(* Logix 5000 project; controller CarbonScout_MK6 vendor 1 type 14 code 154 rev 32.11; software revision 32.00; part 2 of 17 *)
(* tags used below, declared in another part *)
   Inp_PV : REAL;   // Input Signal (process variable) from Sensor
   Inp_PVSrcQ : DINT;   // Input Source and Quality (from Channel object, if available) (enum)
   Inp_PVBad : BOOL;   // 1=PV or I/O Comms Status Bad, 0=OK
   Inp_PVUncertain : BOOL;   // 1=PV Value Not Reliable, 0=OK
   Inp_Sim : BOOL;   // 1=Use simulated PV (Set_SimPV); 0=Use Input (Inp_PV)
   Inp_Reset : BOOL;   // 1=Reset all Alarms requiring reset
   Cfg_NoSubstPV : BOOL;   // 1=Disallow selection of Substitute PV
   Cfg_SetTrack : BOOL;   // 1=PSets track OSets in Oper, OSets track PSets in Prog, 0=no tracking
   Cfg_HasChanObj : BOOL;   // 1=Tells HMI a Channel object (AIChan, etc.) is used for Inp_PV
   Cfg_UseChanSrcQ : BOOL;   // 1=Pass thru connected Channel's SrcQ value, 0=generate SrcQ
   Cfg_PCmdClear : ALIAS FOR Mode.Cfg_PCmdClear;
   Cfg_InpRawMin : REAL;   // Input (unscaled) Minimum for Scaling
   Cfg_InpRawMax : REAL;   // Input (unscaled) Maximum for Scaling
   Cfg_PVEUMin : REAL;   // PV (Output) Minimum for Scaling to EU
   Cfg_PVEUMax : REAL;   // PV (Output) Maximum for Scaling to EU
   Cfg_FiltTC : REAL;   // PV Filter Time Constant (s), 0.0 = unfiltered
   Cfg_HiHiDB : REAL;   // High-High Status Deadband (EU)
   Cfg_HiDB : REAL;   // High Status Deadband (EU)
   Cfg_LoDB : REAL;   // Low Status Deadband (EU)
   Cfg_LoLoDB : REAL;   // Low-Low Status Deadband (EU)
   Cfg_FailHiLim : REAL;   // Out-of-Range (fail) High Limit (EU)
   Cfg_FailLoLim : REAL;   // Out-of-Range (fail) Low Limit (EU)
   Cfg_FailDB : REAL;   // Out-of-Range (fail) High/Low Deadband (EU)
   PSet_Owner : DINT;   // Program Owner Request ID (non-zero) or Release (zero)
   PSet_HiHiLim : REAL;   // Program-Entered High-High Status Threshold (EU)
   PSet_HiLim : REAL;   // Program-Entered High Status Threshold (EU)
   PSet_LoLim : REAL;   // Program-Entered Low Status Threshold (EU)
   PSet_LoLoLim : REAL;   // Program-Entered Low-Low Status Threshold (EU)
   MSet_SubstPV : REAL;   // Maintenance-Entered Substitute PV (EU)
   OSet_HiHiLim : REAL;   // Operator-Entered High-High Status Threshold (EU)
   OSet_HiLim : REAL;   // Operator-Entered High Status Threshold (EU)
   OSet_LoLim : REAL;   // Operator-Entered Low Status Threshold (EU)
   OSet_LoLoLim : REAL;   // Operator-Entered Low-Low Status Threshold (EU)
   Set_SimPV : REAL;   // PV used in Simulation (Inp_Sim=1) (EU)
   PCmd_ClearCapt : BOOL;   // Program Command to Clear the captured min / max PV excursion values
   PCmd_Reset : BOOL;   // Program Command to Reset all Alarms requiring Reset
   PCmd_HiHiAck : ALIAS FOR HiHi.PCmd_Ack;   // Program Command to Acknowledge High-High Alarm
   PCmd_HiAck : ALIAS FOR Hi.PCmd_Ack;   // Program Command to Acknowledge High Alarm
   PCmd_LoAck : ALIAS FOR Lo.PCmd_Ack;   // Program Command to Acknowledge Low Alarm
   PCmd_LoLoAck : ALIAS FOR LoLo.PCmd_Ack;   // Program Command to Acknowledge Low-Low Alarm
   PCmd_FailAck : ALIAS FOR Fail.PCmd_Ack;   // Program Command to Acknowldege Analog Input Failure Alarm
   MCmd_SubstPV : BOOL;   // Maintenance Command to use Substitute PV (override input)
   MCmd_InpPV : BOOL;   // Maintenance Command to use Input PV (normal)
   OCmd_ClearCapt : BOOL;   // Operator Command to Clear the captured min / max PV excursion values
   OCmd_Reset : BOOL;   // Operator Command to Reset all Alarms requiring Reset
   OCmd_ResetAckAll : BOOL;   // Operator Command to Reset and Acknowledge all Alarms
   Val : REAL;   // Analog Value (after Substitute PV, if used)
   Val_InpPV : REAL;   // Analog Input Value (actual, before Substitute PV selection)
   Val_PVMinCapt : REAL;   // Captured PV Minimum (excursion) since last cleared
   Val_PVMaxCapt : REAL;   // Captured PV Maximum (excursion) since last cleared
   Val_PVEUMin : REAL;   // Minimum of scaled range = MIN (Cfg_PVEUMin, Cfg_PVEUMax)
   Val_PVEUMax : REAL;   // Maximum of scaled range = MAX (Cfg_PVEUMin, Cfg_PVEUMax)
   SrcQ_IO : DINT;   // Source and Quality of primary I/O (enumeration)
   SrcQ : DINT;   // Source and Quality of primary Val/Sts (enumeration)
   Val_Fault : DINT;   // Device Fault Status 0=none, 20=Lo, 21=Hi, 24=LoLo, 25=HiHi, 32=Fail, 34=CfgErr
   Val_Owner : DINT;   // Current Object Owner ID (0=not owned)
   Val_Notify : DINT;   // Current Alarm Level and Acknowledgement (enumeration)
   Val_HiHiLim : REAL;   // Current High-High Status Threshold
   Val_HiLim : REAL;   // Current High Status Threshold
   Val_LoLim : REAL;   // Current Low Status Threshold
   Val_LoLoLim : REAL;   // Current Low-Low Status Threshold
   Sts_SubstPV : BOOL;   // 1=Using Substitute PV (Input being overridden)
   Sts_InpPV : BOOL;   // 1=Using Input PV (normal)
   Sts_PVBad : BOOL;   // 1=PV Bad quality or Out of Range
   Sts_PVUncertain : BOOL;   // 1=PV Value is Uncertain (quality)
   Sts_MaintByp : BOOL;   // 1=A Maintenance Bypass is Active, display icon
   Sts_AlmInh : BOOL;   // 1=An Alarm is Shelved, Disabled or Suppressed: display icon
   Sts_Err : BOOL;   // 1=Error in Config (see detail Err_ bits for reason), display icon
   Err_Raw : BOOL;   // 1=Error in Config: Raw Input Scaling Min = Max
   Err_EU : BOOL;   // 1=Error in Config: Scaled EU Min = Max
   Err_Timer : BOOL;   // 1=Error in Config: On Delay, Off Delay, Gate Delay Time Invalid (use 0 to 2147483 s)
   Err_Filt : BOOL;   // 1=Error in Config: PV filter params (RateTime, TC)
   Err_DB : BOOL;   // 1=Error in Config: a Status Deadband is < 0.0
   Err_Alarm : BOOL;   // 1=Error in Config: Alarm Min On Time, Shelf Time, Severity
   Sts_Maint : ALIAS FOR Mode.Sts_Maint;
   Sts_Prog : ALIAS FOR Mode.Sts_Prog;
   Sts_Oper : ALIAS FOR Mode.Sts_Oper;
   Sts_HiHiCmp : ALIAS FOR HiHiGate.Inp;   // PV High-High comparison result 1=High-High
   Sts_HiHi : ALIAS FOR HiHi.Inp;   // 1=Analog Input is above High-High limit
   Sts_HiCmp : ALIAS FOR HiGate.Inp;   // PV High comparison result 1=High
   Sts_Hi : ALIAS FOR Hi.Inp;   // 1=Analog Input is above High limit
   Sts_LoCmp : ALIAS FOR LoGate.Inp;   // PV Low comparison result 1=Low
   Sts_Lo : ALIAS FOR Lo.Inp;   // 1=Analog Input is below Low limit
   Sts_LoLoCmp : ALIAS FOR LoLoGate.Inp;   // PV Low-Low comparison result 1=Low-Low
   Sts_LoLo : ALIAS FOR LoLo.Inp;   // 1=Analog Input is below Low-Low limit
   Sts_FailCmp : ALIAS FOR FailGate.Inp;   // PV Fail comparison result 1=Out of Range
   Sts_Fail : ALIAS FOR Fail.Inp;   // 1=Analog Input is Out of Range or PV Bad
   Rdy_SubstPV : BOOL;   // 1=Ready for MCmd_SubstPV
   Rdy_InpPV : BOOL;   // 1=Ready for MCmd_InpPV
   Rdy_OSet : BOOL;   // 1=Ready to receive OSets (enables data entry fields)
   P_AIn : BOOL;   // Unique Parameter Name for auto - discovery
   LoLo : P_Alarm;   // Low-Low Alarm
   Lo : P_Alarm;   // Low Alarm
   Hi : P_Alarm;   // High Alarm
   HiHi : P_Alarm;   // High-High Alarm
   Mode : P_Mode;   // Analog Input Mode Selection
   Cfg_Tag : STRING_12;   // Tagname for display on HMI
   Cfg_Label : STRING_12;   // Label for graphic symbol displayed on HMI
   Cfg_Desc : STRING_20;   // Description for display on HMI
   Fail : P_Alarm;   // Analog Input Failure Alarm (bad quality or out of range)
   Wrk_Notify : DINT;   // Buffer for building Val_Notify
   Wrk_SrcQ : DINT;   // Register for building Source / Quality enumeration
   Wrk_Fault : DINT;   // Buffer for building Val_Fault
   Wrk_SubstPV : BOOL;   // Internal flag: Using Substitute PV
   Wrk_UnfiltPV : REAL;   // Unfiltered PV, input to 1st order filter
   Wrk_Alpha : REAL;   // Filter multiplier = (1 / (1+TC/dT) )
   Wrk_ScanT : TIMER;   // Scan Timer (milliseconds, always runs)
   Wrk_ScanTime : REAL;   // Time since this instance was last scanned
   Wrk_FiltPV : REAL;   // Filtered PV
   Wrk_ValidONS : BOOL;   // Selected PV goes from Infinite or Not a Number to VALID
   Wrk_SelPVDINT : DINT;   // Selected PV check for Infinite or Non A Number
   Wrk_SelPVInfNaN : BOOL;   // Selected PV (Input or Substitute) is Infinite or NaN
   Wrk_Fail : BOOL;   // Internal flag: Fail Status
   Wrk_LoLo : BOOL;   // Internal flag: Low-Low Status
   Wrk_Lo : BOOL;   // Internal flag: Low Status
   Wrk_Hi : BOOL;   // Internal flag: High Status
   Wrk_HiHi : BOOL;   // Internal flag: High-High Status
   FailGate : P_Gate;   // Fail Alarm Gate / Delay Block
   LoLoGate : P_Gate;   // Low-Low Alarm Gate / Delay Block
   LoGate : P_Gate;   // Low Alarm Gate / Delay Block
   HiHiGate : P_Gate;   // High-High Alarm Gate / Delay Block
   HiGate : P_Gate;   // High Alarm Gate / Delay Block
   Wrk_InpInfNaN : BOOL;   // Input is Infinite or Not a Number
   Wrk_InpDINT : DINT;   // Input REAL bit pattern as a DINT (check for Inf/NaN)
   Wrk_InpFail : BOOL;   // Input Fail: out of range
   Simulation : DINT;
   test : DINT;
(* P_AIn, continued *)

ROUTINE Logic   (* ladder *)
// Normal Scan - PV is scaled and alarms are generated
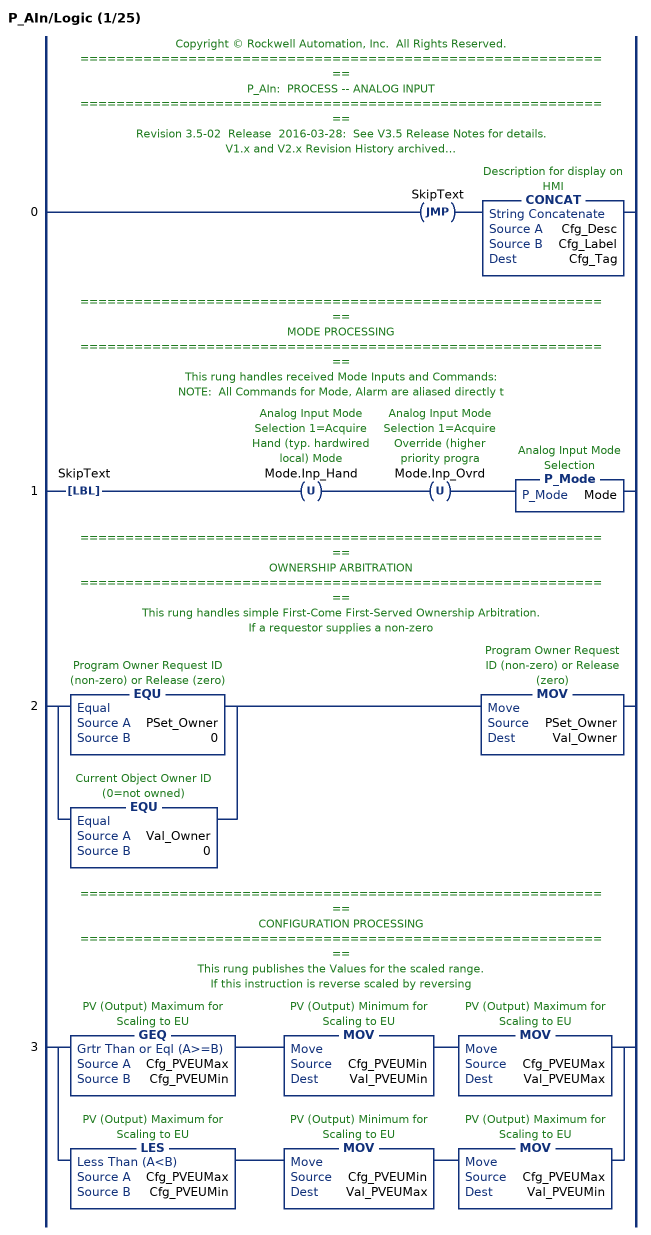
   // Copyright © Rockwell Automation, Inc.  All Rights Reserved.
   // ============================================================
   // P_AIn:  PROCESS -- ANALOG INPUT
   // ============================================================
   // Revision 3.5-02  Release  2016-03-28:  See V3.5 Release Notes for details.
   // V1.x and V2.x Revision History archived.
   // V3.0-00  2013-06-30:  Uses P_Gate, P_Alarm, P_Mode V3.0.
   // Added Inf_Lib, navigation to Channel obj.
   // V3.0-01  2013-07-30:  Modified Parameter descriptions only.
   // V3.0-02  2013-09-03:  Modified Parameter descriptions only.
   // V3.0-03  2013-10-30:  Corrected Parameter descriptions and default
   // configuration values for alarms only.
   // V3.0-04  2014-04-04:   Improved handling of Inf/NaN to avoid Minor Faults.
   // V3.1-00  2014-07-08:  Modified to use P_Alarm, P_Mode V3.1, add SrcQ enums.
   // Modified to consistently use alias tag names.
   // V3.1-01  2014-09-03:  Inp_PVSrcQ pulled into all bad/uncertain logic.
   // Using P_Alarm, P_Gate, P_Mode V3.1-01.
   // V3.1-02  2014-09-30:  Unchanged, but using P_Alarm V3.1-02.
   // V3.1-05  2016-01-22:  Added check of SrcQ >= 32 for Val_Fault.
   // Changed default values of min, max capture. Modified to
   // handle on-delay near status thresholds properly.
   // V3.5-01  2016-01-29:  Unchanged, using P_Alarm, P_Gate V3.5-01.
   // V3.5-02  2016-03-28:  Added Cfg_UseChanSrcQ to make SrcQ use
   // independent of Cfg_HasChanObj, which is for navigation only.
   // ============================================================
   // This Instruction monitors an Analog Input from a flow, level, pressure,
   // temperature, or any other analog sensor, and provides:
   // *  Scaling, from Input (Raw) to PV (Engineering) Units
   // *  High-High, High, Low and Low-Low Status and Alarms, with Gate
   // inputs and configurable on-delay, off-delay and gate delay times
   // *  Monitoring of bad/uncertain PV status, floating point exceptions
   // and out-of-range conditions, with PV Fail alarm
   // *  Setting of a simulated input signal for process simulation
   // *  Capturing of the lowest and highest PV excursion values
   // *  Program and Operator Settings for Status Thresholds
   // *  Configurable threshold deadbands and out of range limits
   // *  Maintenance Commands to allow manual override of the input signal (Substitute PV)
   // Modes are provided by a P_Mode AOI instance.
   // Alarms are provided by P_Alarm AOI instances.
   // Status gating provided by P_Gate AOI instances.
   // Modes of operation: Operator, Program, Maintenance
   // ============================================================
   // SHOW LOCAL STRINGS
   // ============================================================
   // The STRINGs containing the text associated with each instance of this
   // instruction cannot be Input or Output Parameters, because STRINGs are not
   //  'atomic' types. (Inputs and Outputs must be SINT, INT, DINT, REAL, or BOOL.)
   // In order to make it easier to find and configure these STRINGs, this rung
   // was added.  THE JMP (and the LBL on the following rung)
   // MUST NOT BE REMOVED!!!
   // To view the STRINGs, go to the instruction instance (in LD or FBD), RIGHT-click
   // to bring up the context menu and select "Open Instruction Logic".
   // This rung will appear with the STRING values for the selected instance.
   // You may double-click the STRING values here to modify them as well.
   // #####  V3.0-00  2013-06-30:  Added Inf_Lib  #####
   0: JMP(SkipText)CONCAT(Cfg_Desc,Cfg_Label,Cfg_Tag);
   // ============================================================
   // MODE PROCESSING
   // ============================================================
   // This rung handles received Mode Inputs and Commands:
   // NOTE:  All Commands for Mode, Alarm are aliased directly t
   1: LBL(SkipText)OTU(Mode.Inp_Hand)OTU(Mode.Inp_Ovrd)P_Mode(Mode);
   // ============================================================
   // OWNERSHIP ARBITRATION
   // ============================================================
   // This rung handles simple First-Come First-Served Ownership Arbitration.
   // If a requestor supplies a non-zero
   2: [EQU(PSet_Owner,0) ,EQU(Val_Owner,0) ]MOV(PSet_Owner,Val_Owner);
   // ============================================================
   // CONFIGURATION PROCESSING
   // ============================================================
   // This rung publishes the Values for the scaled range.
   // If this instruction is reverse scaled by reversing
   3: [GEQ(Cfg_PVEUMax,Cfg_PVEUMin) MOV(Cfg_PVEUMin,Val_PVEUMin) MOV(Cfg_PVEUMax,Val_PVEUMax) ,LES(Cfg_PVEUMax,Cfg_PVEUMin) MOV(Cfg_PVEUMin,Val_PVEUMax) MOV(Cfg_PVEUMax,Val_PVEUMin) ];
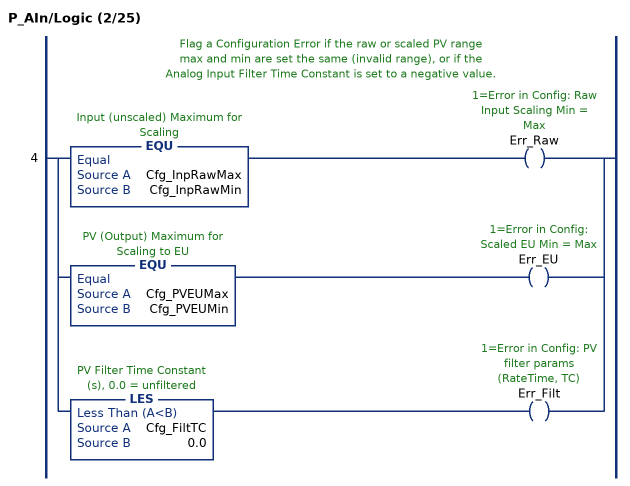
   // Flag a Configuration Error if the raw or scaled PV range
   // max and min are set the same (invalid range), or if the
   // Analog Input Filter Time Constant is set to a negative value.
   4: [EQU(Cfg_InpRawMax,Cfg_InpRawMin) OTE(Err_Raw) ,EQU(Cfg_PVEUMax,Cfg_PVEUMin) OTE(Err_EU) ,LES(Cfg_FiltTC,0.0) OTE(Err_Filt) ];
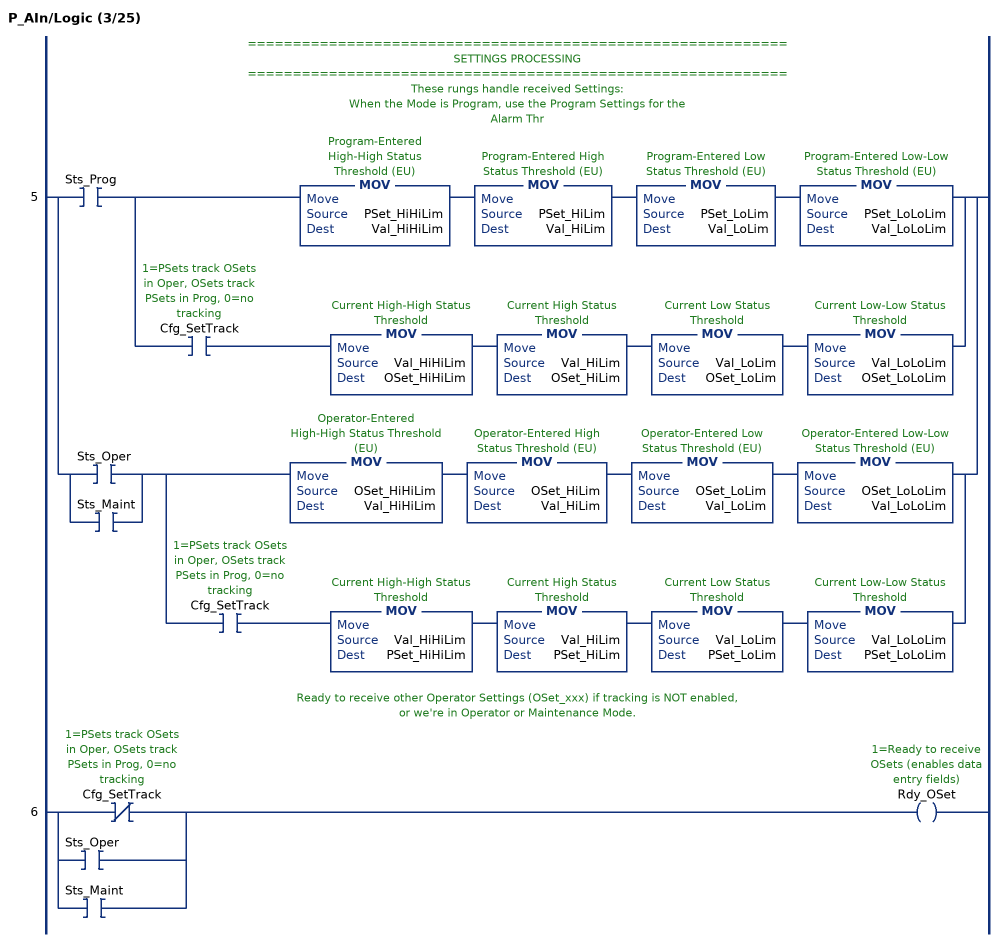
   // ============================================================
   // SETTINGS PROCESSING
   // ============================================================
   // These rungs handle received Settings:
   // When the Mode is Program, use the Program Settings for the
   // Alarm Thr
   5: [XIC(Sts_Prog) [MOV(PSet_HiHiLim,Val_HiHiLim) MOV(PSet_HiLim,Val_HiLim) MOV(PSet_LoLim,Val_LoLim) MOV(PSet_LoLoLim,Val_LoLoLim) ,XIC(Cfg_SetTrack) MOV(Val_HiHiLim,OSet_HiHiLim) MOV(Val_HiLim,OSet_HiLim) MOV(Val_LoLim,OSet_LoLim) MOV(Val_LoLoLim,OSet_LoLoLim) ] ,[XIC(Sts_Oper) ,XIC(Sts_Maint) ] [MOV(OSet_HiHiLim,Val_HiHiLim) MOV(OSet_HiLim,Val_HiLim) MOV(OSet_LoLim,Val_LoLim) MOV(OSet_LoLoLim,Val_LoLoLim) ,XIC(Cfg_SetTrack) MOV(Val_HiHiLim,PSet_HiHiLim) MOV(Val_HiLim,PSet_HiLim) MOV(Val_LoLim,PSet_LoLim) MOV(Val_LoLoLim,PSet_LoLoLim) ] ];
   // Ready to receive other Operator Settings (OSet_xxx) if tracking is NOT enabled,
   // or we're in Operator or Maintenance Mode.
   6: [XIO(Cfg_SetTrack) ,XIC(Sts_Oper) ,XIC(Sts_Maint) ]OTE(Rdy_OSet);
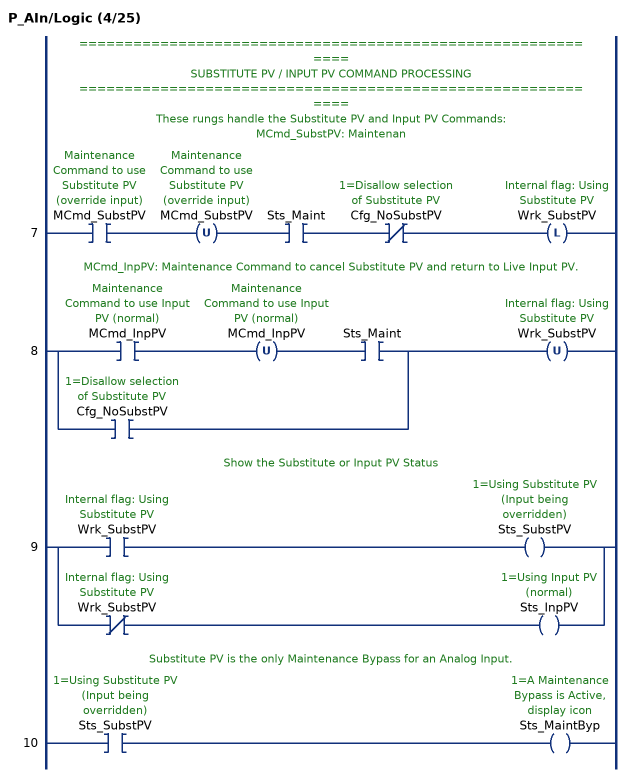
   // ============================================================
   // SUBSTITUTE PV / INPUT PV COMMAND PROCESSING
   // ============================================================
   // These rungs handle the Substitute PV and Input PV Commands:
   // MCmd_SubstPV: Maintenan
   7: XIC(MCmd_SubstPV)OTU(MCmd_SubstPV)XIC(Sts_Maint)XIO(Cfg_NoSubstPV)OTL(Wrk_SubstPV);
   // MCmd_InpPV: Maintenance Command to cancel Substitute PV and return to Live Input PV.
   8: [XIC(MCmd_InpPV) OTU(MCmd_InpPV) XIC(Sts_Maint) ,XIC(Cfg_NoSubstPV) ]OTU(Wrk_SubstPV);
   // Show the Substitute or Input PV Status
   9: [XIC(Wrk_SubstPV) OTE(Sts_SubstPV) ,XIO(Wrk_SubstPV) OTE(Sts_InpPV) ];
   // Substitute PV is the only Maintenance Bypass for an Analog Input.
   10: XIC(Sts_SubstPV)OTE(Sts_MaintByp);
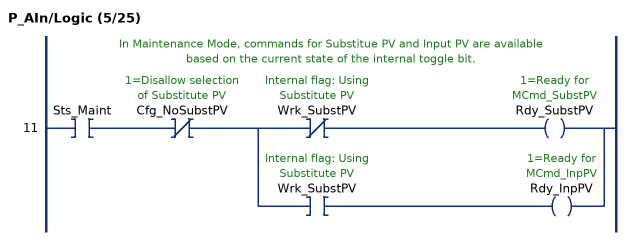
   // In Maintenance Mode, commands for Substitue PV and Input PV are available
   // based on the current state of the internal toggle bit.
   11: XIC(Sts_Maint)XIO(Cfg_NoSubstPV)[XIO(Wrk_SubstPV) OTE(Rdy_SubstPV) ,XIC(Wrk_SubstPV) OTE(Rdy_InpPV) ];
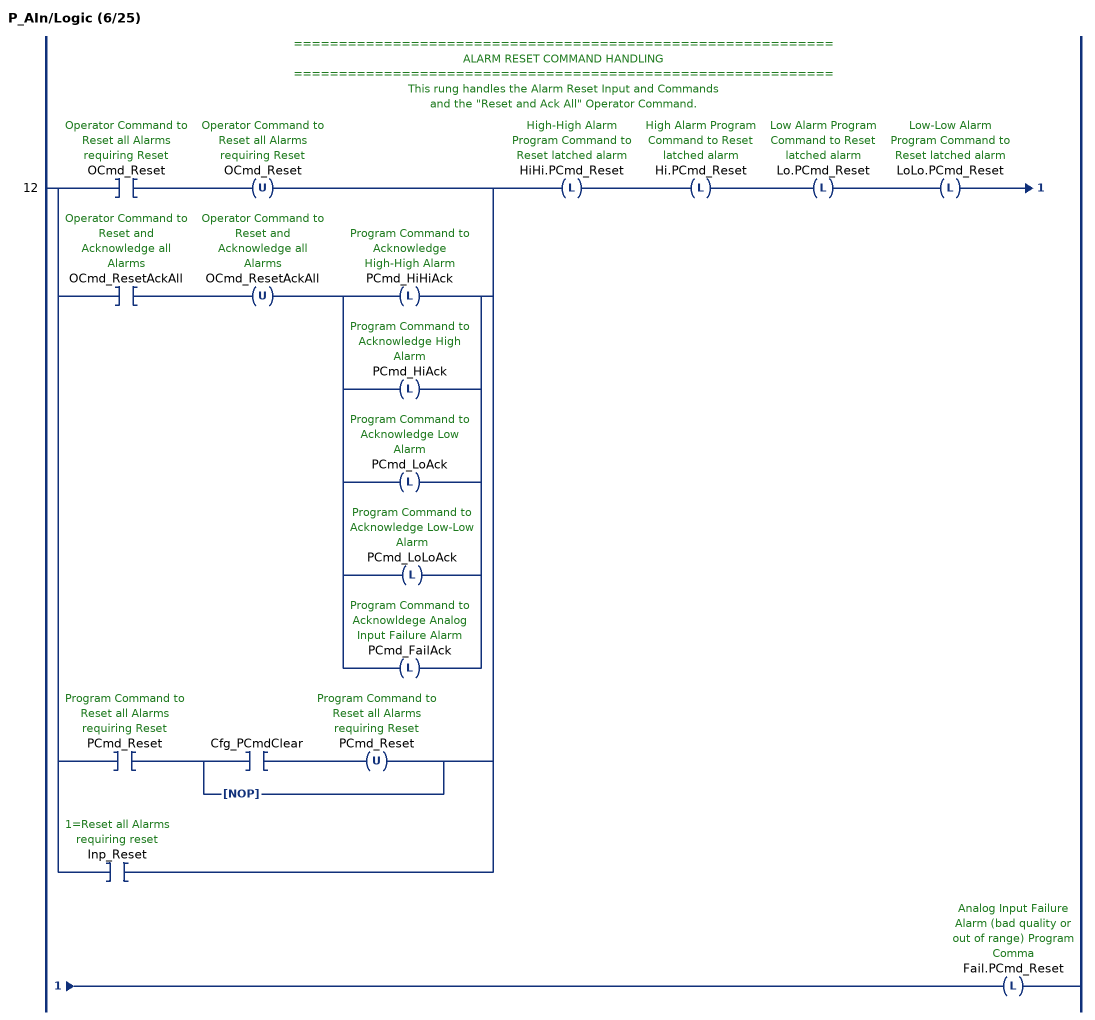
   // ============================================================
   // ALARM RESET COMMAND HANDLING
   // ============================================================
   // This rung handles the Alarm Reset Input and Commands
   // and the "Reset and Ack All" Operator Command.
   12: [XIC(OCmd_Reset) OTU(OCmd_Reset) ,XIC(OCmd_ResetAckAll) OTU(OCmd_ResetAckAll) [OTL(PCmd_HiHiAck) ,OTL(PCmd_HiAck) ,OTL(PCmd_LoAck) ,OTL(PCmd_LoLoAck) ,OTL(PCmd_FailAck) ] ,XIC(PCmd_Reset) [XIC(Cfg_PCmdClear) OTU(PCmd_Reset) ,NOP() ] ,XIC(Inp_Reset) ]OTL(HiHi.PCmd_Reset)OTL(Hi.PCmd_Reset)OTL(Lo.PCmd_Reset)OTL(LoLo.PCmd_Reset)OTL(Fail.PCmd_Reset);
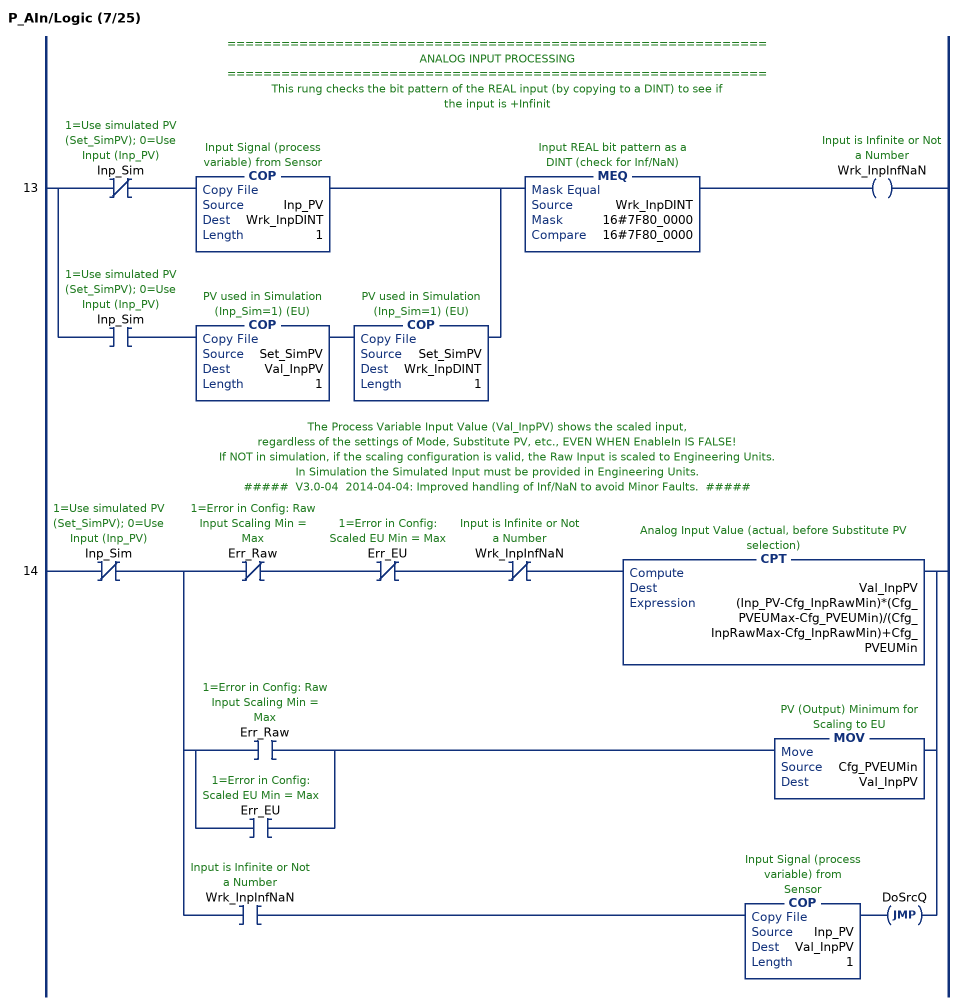
   // ============================================================
   // ANALOG INPUT PROCESSING
   // ============================================================
   // This rung checks the bit pattern of the REAL input (by copying to a DINT) to see if
   // the input is +Infinit
   13: [XIO(Inp_Sim) COP(Inp_PV,Wrk_InpDINT,1) ,XIC(Inp_Sim) COP(Set_SimPV,Val_InpPV,1) COP(Set_SimPV,Wrk_InpDINT,1) ]MEQ(Wrk_InpDINT,16#7F80_0000,16#7F80_0000)OTE(Wrk_InpInfNaN);
   // The Process Variable Input Value (Val_InpPV) shows the scaled input,
   // regardless of the settings of Mode, Substitute PV, etc., EVEN WHEN EnableIn IS FALSE!
   // If NOT in simulation, if the scaling configuration is valid, the Raw Input is scaled to Engineering Units.
   // In Simulation the Simulated Input must be provided in Engineering Units.
   // #####  V3.0-04  2014-04-04: Improved handling of Inf/NaN to avoid Minor Faults.  #####
   14: XIO(Inp_Sim)[XIO(Err_Raw) XIO(Err_EU) XIO(Wrk_InpInfNaN) CPT(Val_InpPV,(Inp_PV-Cfg_InpRawMin)*(Cfg_PVEUMax-Cfg_PVEUMin)/(Cfg_InpRawMax-Cfg_InpRawMin)+Cfg_PVEUMin) ,[XIC(Err_Raw) ,XIC(Err_EU) ] MOV(Cfg_PVEUMin,Val_InpPV) ,XIC(Wrk_InpInfNaN) COP(Inp_PV,Val_InpPV,1) JMP(DoSrcQ) ];
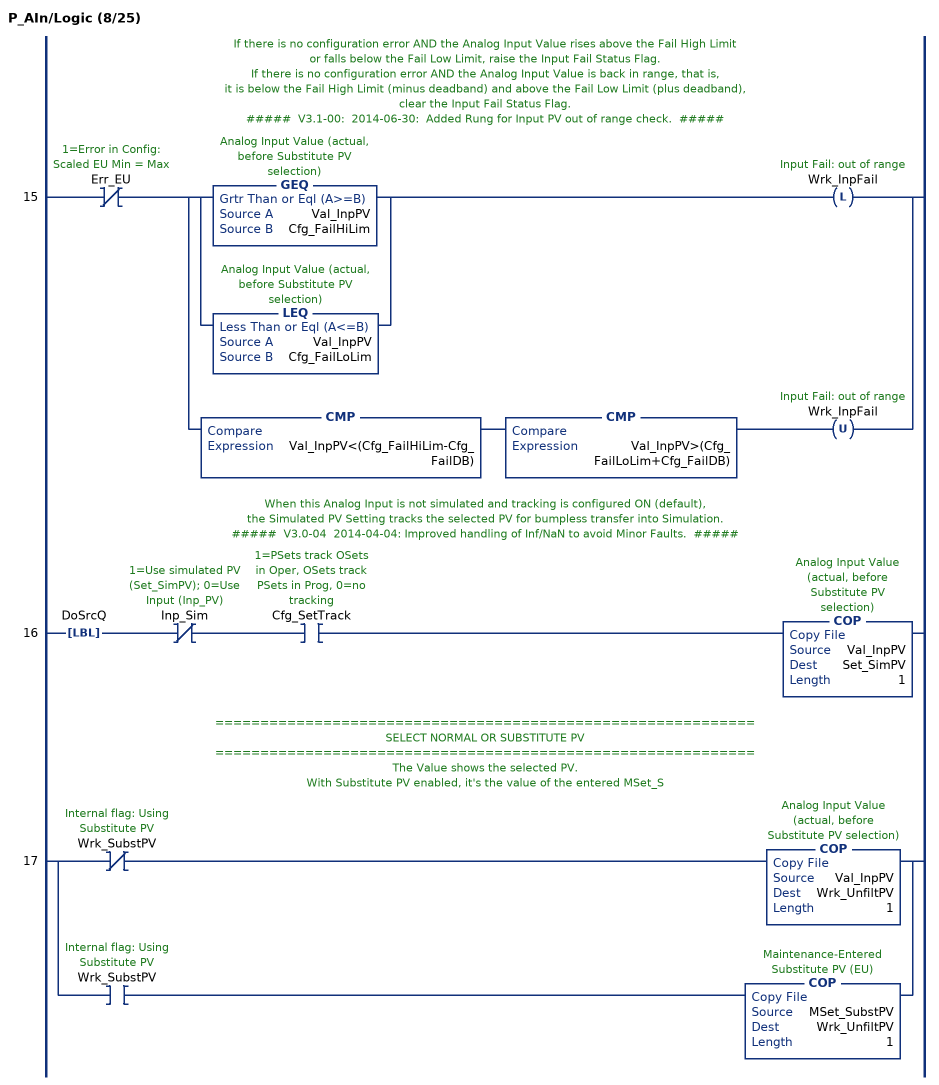
   // If there is no configuration error AND the Analog Input Value rises above the Fail High Limit
   // or falls below the Fail Low Limit, raise the Input Fail Status Flag.
   // If there is no configuration error AND the Analog Input Value is back in range, that is,
   // it is below the Fail High Limit (minus deadband) and above the Fail Low Limit (plus deadband),
   // clear the Input Fail Status Flag.
   // #####  V3.1-00:  2014-06-30:  Added Rung for Input PV out of range check.  #####
   15: XIO(Err_EU)[[GEQ(Val_InpPV,Cfg_FailHiLim) ,LEQ(Val_InpPV,Cfg_FailLoLim) ] OTL(Wrk_InpFail) ,CMP(Val_InpPV<(Cfg_FailHiLim-Cfg_FailDB)) CMP(Val_InpPV>(Cfg_FailLoLim+Cfg_FailDB)) OTU(Wrk_InpFail) ];
   // When this Analog Input is not simulated and tracking is configured ON (default),
   // the Simulated PV Setting tracks the selected PV for bumpless transfer into Simulation.
   // #####  V3.0-04  2014-04-04: Improved handling of Inf/NaN to avoid Minor Faults.  #####
   16: LBL(DoSrcQ)XIO(Inp_Sim)XIC(Cfg_SetTrack)COP(Val_InpPV,Set_SimPV,1);
   // ============================================================
   // SELECT NORMAL OR SUBSTITUTE PV
   // ============================================================
   // The Value shows the selected PV.
   // With Substitute PV enabled, it's the value of the entered MSet_S
   17: [XIO(Wrk_SubstPV) COP(Val_InpPV,Wrk_UnfiltPV,1) ,XIC(Wrk_SubstPV) COP(MSet_SubstPV,Wrk_UnfiltPV,1) ];
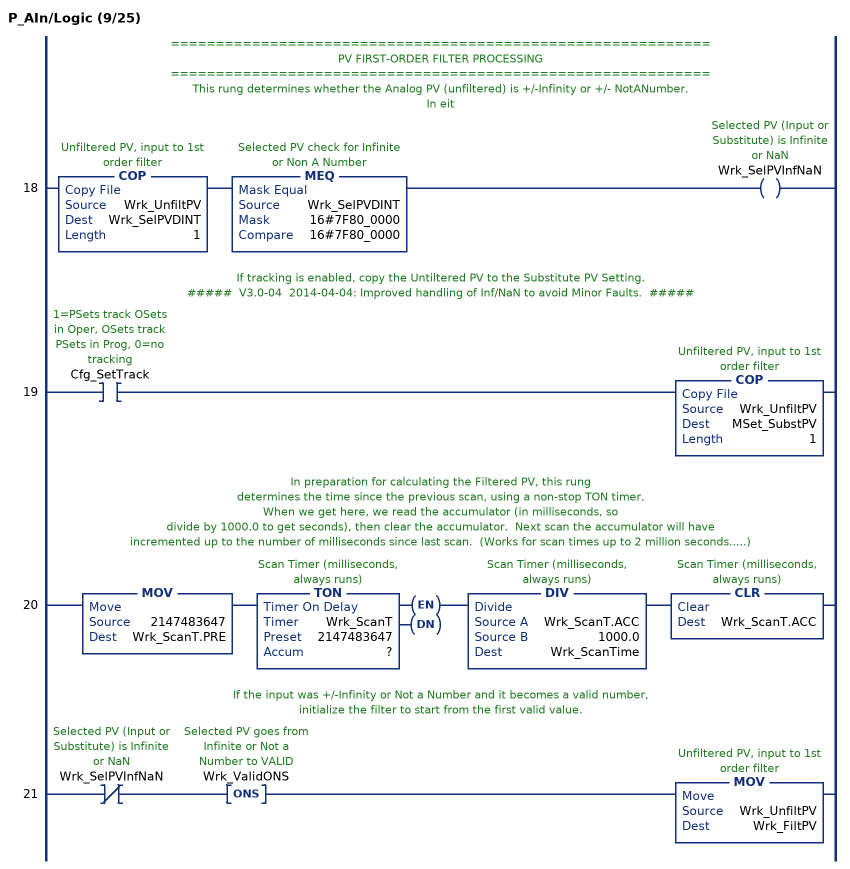
   // ============================================================
   // PV FIRST-ORDER FILTER PROCESSING
   // ============================================================
   // This rung determines whether the Analog PV (unfiltered) is +/-Infinity or +/- NotANumber.
   // In eit
   18: COP(Wrk_UnfiltPV,Wrk_SelPVDINT,1)MEQ(Wrk_SelPVDINT,16#7F80_0000,16#7F80_0000)OTE(Wrk_SelPVInfNaN);
   // If tracking is enabled, copy the Untiltered PV to the Substitute PV Setting.
   // #####  V3.0-04  2014-04-04: Improved handling of Inf/NaN to avoid Minor Faults.  #####
   19: XIC(Cfg_SetTrack)COP(Wrk_UnfiltPV,MSet_SubstPV,1);
   // In preparation for calculating the Filtered PV, this rung
   // determines the time since the previous scan, using a non-stop TON timer.
   // When we get here, we read the accumulator (in milliseconds, so
   // divide by 1000.0 to get seconds), then clear the accumulator.  Next scan the accumulator will have
   // incremented up to the number of milliseconds since last scan.  (Works for scan times up to 2 million seconds.....)
   20: MOV(2147483647,Wrk_ScanT.PRE)TON(Wrk_ScanT,?,?)DIV(Wrk_ScanT.ACC,1000.0,Wrk_ScanTime)CLR(Wrk_ScanT.ACC);
   // If the input was +/-Infinity or Not a Number and it becomes a valid number,
   // initialize the filter to start from the first valid value.
   21: XIO(Wrk_SelPVInfNaN)ONS(Wrk_ValidONS)MOV(Wrk_UnfiltPV,Wrk_FiltPV);
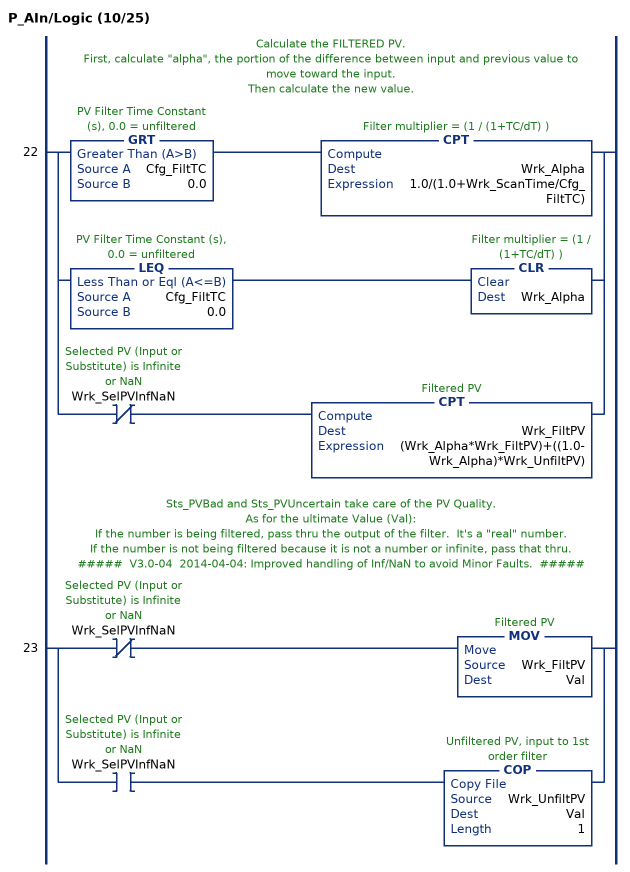
   // Calculate the FILTERED PV.
   // First, calculate "alpha", the portion of the difference between input and previous value to move toward the input.
   // Then calculate the new value.
   22: [GRT(Cfg_FiltTC,0.0) CPT(Wrk_Alpha,1.0/(1.0+Wrk_ScanTime/Cfg_FiltTC)) ,LEQ(Cfg_FiltTC,0.0) CLR(Wrk_Alpha) ,XIO(Wrk_SelPVInfNaN) CPT(Wrk_FiltPV,(Wrk_Alpha*Wrk_FiltPV)+((1.0-Wrk_Alpha)*Wrk_UnfiltPV)) ];
   // Sts_PVBad and Sts_PVUncertain take care of the PV Quality.
   // As for the ultimate Value (Val):
   // If the number is being filtered, pass thru the output of the filter.  It's a "real" number.
   // If the number is not being filtered because it is not a number or infinite, pass that thru.
   // #####  V3.0-04  2014-04-04: Improved handling of Inf/NaN to avoid Minor Faults.  #####
   23: [XIO(Wrk_SelPVInfNaN) MOV(Wrk_FiltPV,Val) ,XIC(Wrk_SelPVInfNaN) COP(Wrk_UnfiltPV,Val,1) ];
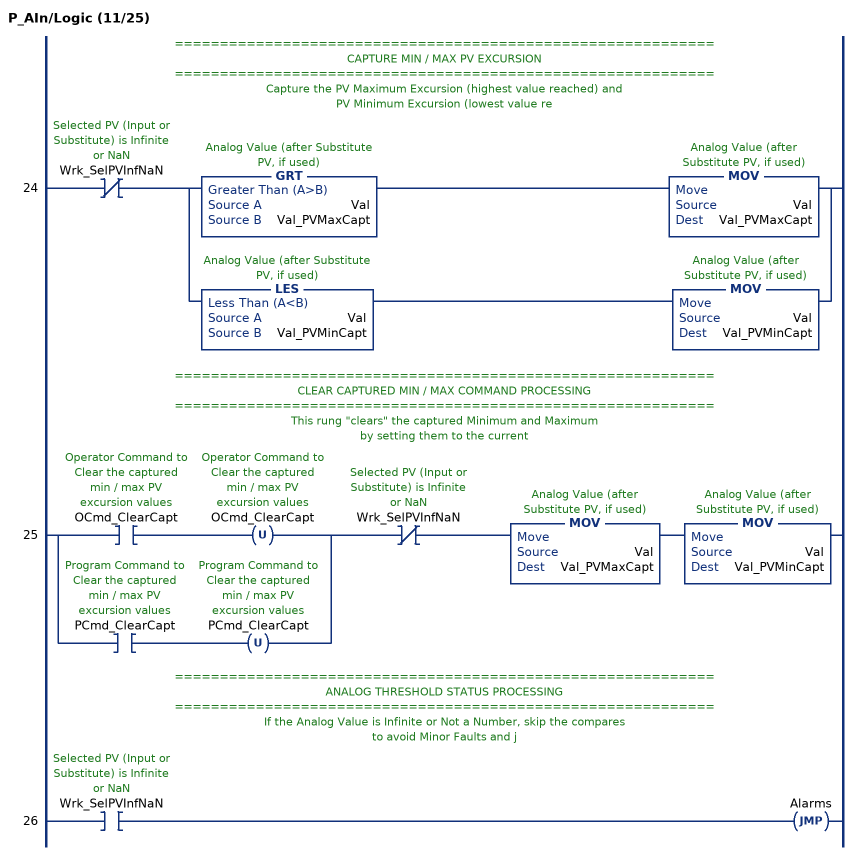
   // ============================================================
   // CAPTURE MIN / MAX PV EXCURSION
   // ============================================================
   // Capture the PV Maximum Excursion (highest value reached) and
   // PV Minimum Excursion (lowest value re
   24: XIO(Wrk_SelPVInfNaN)[GRT(Val,Val_PVMaxCapt) MOV(Val,Val_PVMaxCapt) ,LES(Val,Val_PVMinCapt) MOV(Val,Val_PVMinCapt) ];
   // ============================================================
   // CLEAR CAPTURED MIN / MAX COMMAND PROCESSING
   // ============================================================
   // This rung "clears" the captured Minimum and Maximum
   // by setting them to the current
   25: [XIC(OCmd_ClearCapt) OTU(OCmd_ClearCapt) ,XIC(PCmd_ClearCapt) OTU(PCmd_ClearCapt) ]XIO(Wrk_SelPVInfNaN)MOV(Val,Val_PVMaxCapt)MOV(Val,Val_PVMinCapt);
   // ============================================================
   // ANALOG THRESHOLD STATUS PROCESSING
   // ============================================================
   // If the Analog Value is Infinite or Not a Number, skip the compares
   // to avoid Minor Faults and j
   26: XIC(Wrk_SelPVInfNaN)JMP(Alarms);
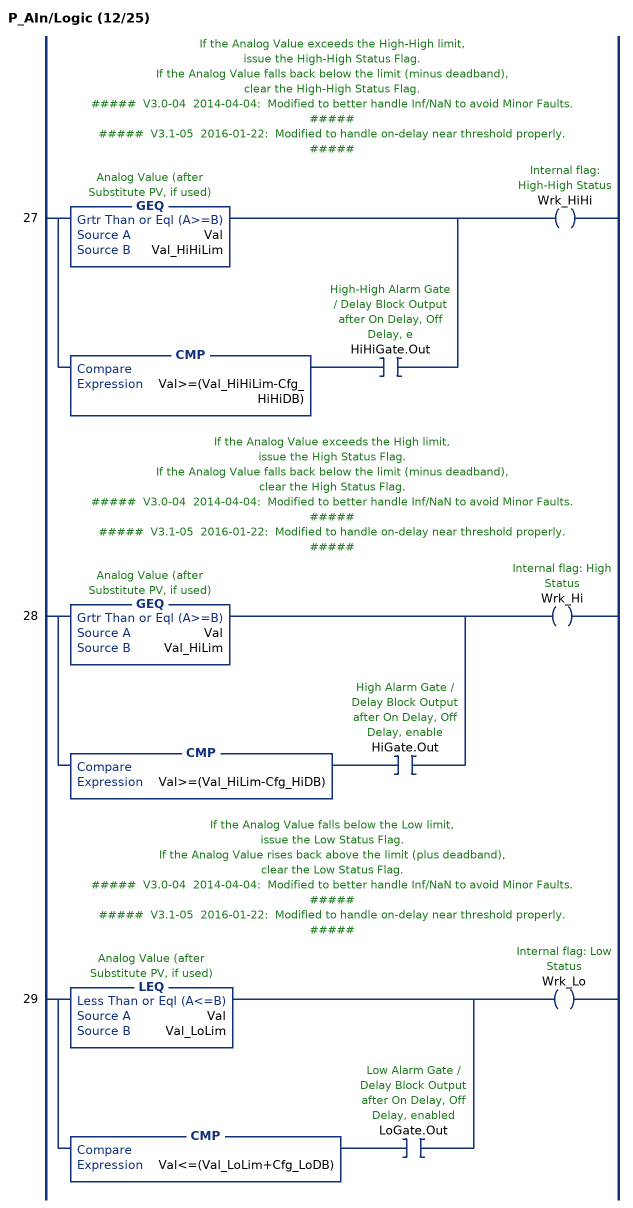
   // If the Analog Value exceeds the High-High limit,
   // issue the High-High Status Flag.
   // If the Analog Value falls back below the limit (minus deadband),
   // clear the High-High Status Flag.
   // #####  V3.0-04  2014-04-04:  Modified to better handle Inf/NaN to avoid Minor Faults.  #####
   // #####  V3.1-05  2016-01-22:  Modified to handle on-delay near threshold properly.  #####
   27: [GEQ(Val,Val_HiHiLim) ,CMP(Val>=(Val_HiHiLim-Cfg_HiHiDB)) XIC(HiHiGate.Out) ]OTE(Wrk_HiHi);
   // If the Analog Value exceeds the High limit,
   // issue the High Status Flag.
   // If the Analog Value falls back below the limit (minus deadband),
   // clear the High Status Flag.
   // #####  V3.0-04  2014-04-04:  Modified to better handle Inf/NaN to avoid Minor Faults.  #####
   // #####  V3.1-05  2016-01-22:  Modified to handle on-delay near threshold properly.  #####
   28: [GEQ(Val,Val_HiLim) ,CMP(Val>=(Val_HiLim-Cfg_HiDB)) XIC(HiGate.Out) ]OTE(Wrk_Hi);
   // If the Analog Value falls below the Low limit,
   // issue the Low Status Flag.
   // If the Analog Value rises back above the limit (plus deadband),
   // clear the Low Status Flag.
   // #####  V3.0-04  2014-04-04:  Modified to better handle Inf/NaN to avoid Minor Faults.  #####
   // #####  V3.1-05  2016-01-22:  Modified to handle on-delay near threshold properly.  #####
   29: [LEQ(Val,Val_LoLim) ,CMP(Val<=(Val_LoLim+Cfg_LoDB)) XIC(LoGate.Out) ]OTE(Wrk_Lo);
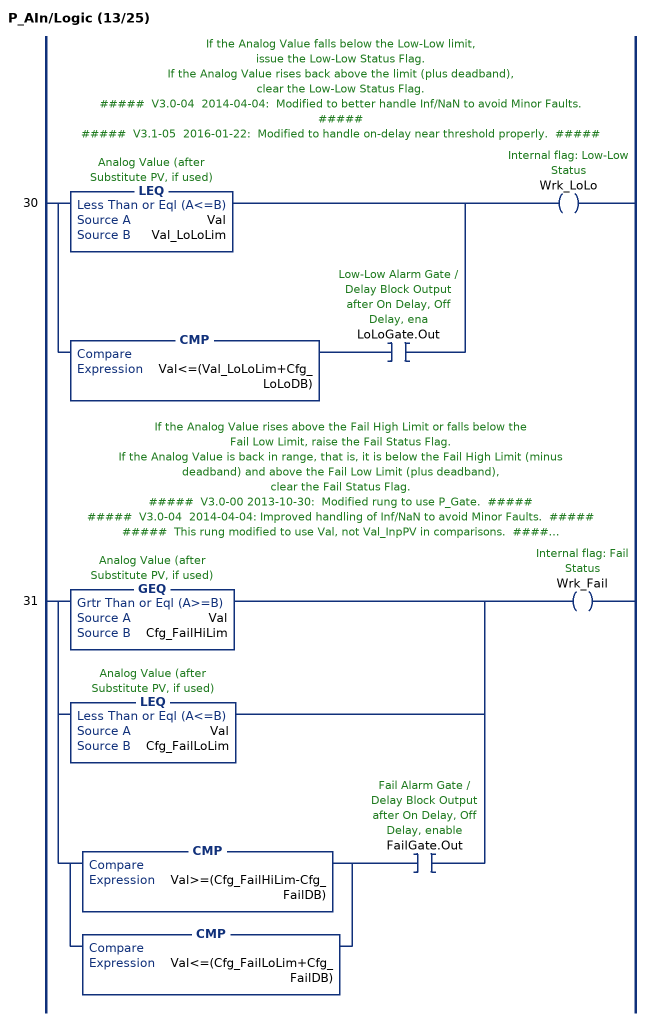
   // If the Analog Value falls below the Low-Low limit,
   // issue the Low-Low Status Flag.
   // If the Analog Value rises back above the limit (plus deadband),
   // clear the Low-Low Status Flag.
   // #####  V3.0-04  2014-04-04:  Modified to better handle Inf/NaN to avoid Minor Faults.  #####
   // #####  V3.1-05  2016-01-22:  Modified to handle on-delay near threshold properly.  #####
   30: [LEQ(Val,Val_LoLoLim) ,CMP(Val<=(Val_LoLoLim+Cfg_LoLoDB)) XIC(LoLoGate.Out) ]OTE(Wrk_LoLo);
   // If the Analog Value rises above the Fail High Limit or falls below the
   // Fail Low Limit, raise the Fail Status Flag.
   // If the Analog Value is back in range, that is, it is below the Fail High Limit (minus
   // deadband) and above the Fail Low Limit (plus deadband),
   // clear the Fail Status Flag.
   // #####  V3.0-00 2013-10-30:  Modified rung to use P_Gate.  #####
   // #####  V3.0-04  2014-04-04: Improved handling of Inf/NaN to avoid Minor Faults.  #####
   // #####  This rung modified to use Val, not Val_InpPV in comparisons.  #####
   // #####  V3.1-05  2016-01-22:  Modified to handle on-delay near threshold properly.  #####
   31: [[GEQ(Val,Cfg_FailHiLim) ,LEQ(Val,Cfg_FailLoLim) ] ,[CMP(Val>=(Cfg_FailHiLim-Cfg_FailDB)) ,CMP(Val<=(Cfg_FailLoLim+Cfg_FailDB)) ] XIC(FailGate.Out) ]OTE(Wrk_Fail);
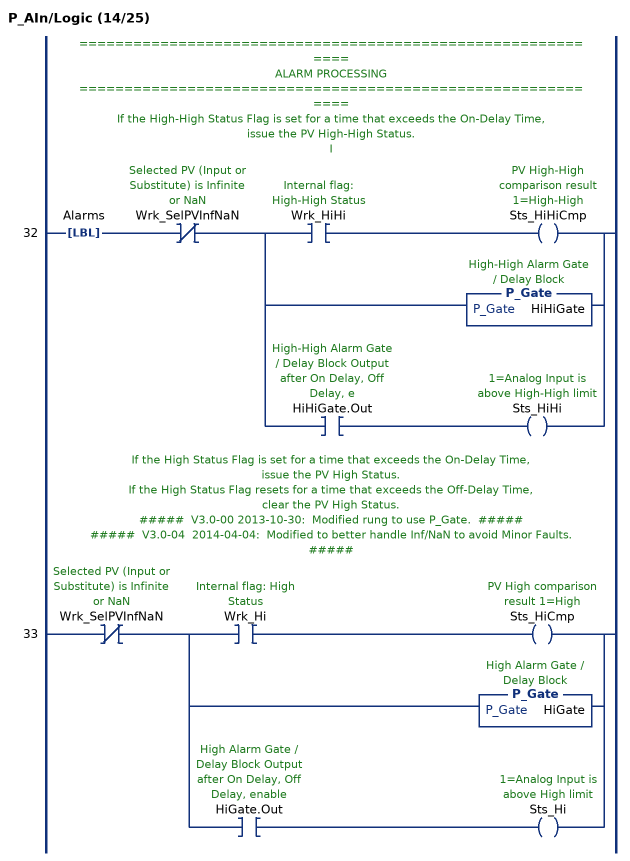
   // ============================================================
   // ALARM PROCESSING
   // ============================================================
   // If the High-High Status Flag is set for a time that exceeds the On-Delay Time,
   // issue the PV High-High Status.
   // I
   32: LBL(Alarms)XIO(Wrk_SelPVInfNaN)[XIC(Wrk_HiHi) OTE(Sts_HiHiCmp) ,P_Gate(HiHiGate) ,XIC(HiHiGate.Out) OTE(Sts_HiHi) ];
   // If the High Status Flag is set for a time that exceeds the On-Delay Time,
   // issue the PV High Status.
   // If the High Status Flag resets for a time that exceeds the Off-Delay Time,
   // clear the PV High Status.
   // #####  V3.0-00 2013-10-30:  Modified rung to use P_Gate.  #####
   // #####  V3.0-04  2014-04-04:  Modified to better handle Inf/NaN to avoid Minor Faults.  #####
   33: XIO(Wrk_SelPVInfNaN)[XIC(Wrk_Hi) OTE(Sts_HiCmp) ,P_Gate(HiGate) ,XIC(HiGate.Out) OTE(Sts_Hi) ];
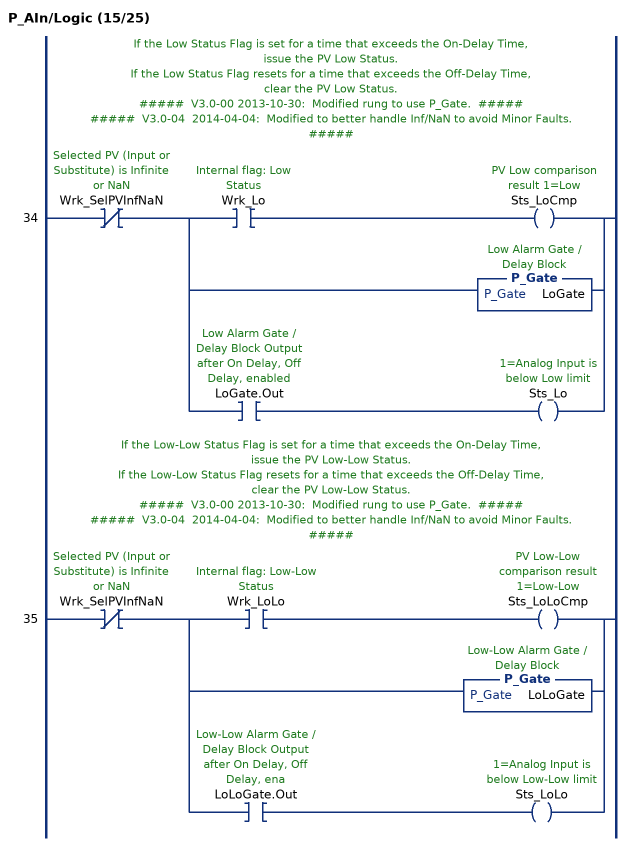
   // If the Low Status Flag is set for a time that exceeds the On-Delay Time,
   // issue the PV Low Status.
   // If the Low Status Flag resets for a time that exceeds the Off-Delay Time,
   // clear the PV Low Status.
   // #####  V3.0-00 2013-10-30:  Modified rung to use P_Gate.  #####
   // #####  V3.0-04  2014-04-04:  Modified to better handle Inf/NaN to avoid Minor Faults.  #####
   34: XIO(Wrk_SelPVInfNaN)[XIC(Wrk_Lo) OTE(Sts_LoCmp) ,P_Gate(LoGate) ,XIC(LoGate.Out) OTE(Sts_Lo) ];
   // If the Low-Low Status Flag is set for a time that exceeds the On-Delay Time,
   // issue the PV Low-Low Status.
   // If the Low-Low Status Flag resets for a time that exceeds the Off-Delay Time,
   // clear the PV Low-Low Status.
   // #####  V3.0-00 2013-10-30:  Modified rung to use P_Gate.  #####
   // #####  V3.0-04  2014-04-04:  Modified to better handle Inf/NaN to avoid Minor Faults.  #####
   35: XIO(Wrk_SelPVInfNaN)[XIC(Wrk_LoLo) OTE(Sts_LoLoCmp) ,P_Gate(LoLoGate) ,XIC(LoLoGate.Out) OTE(Sts_LoLo) ];
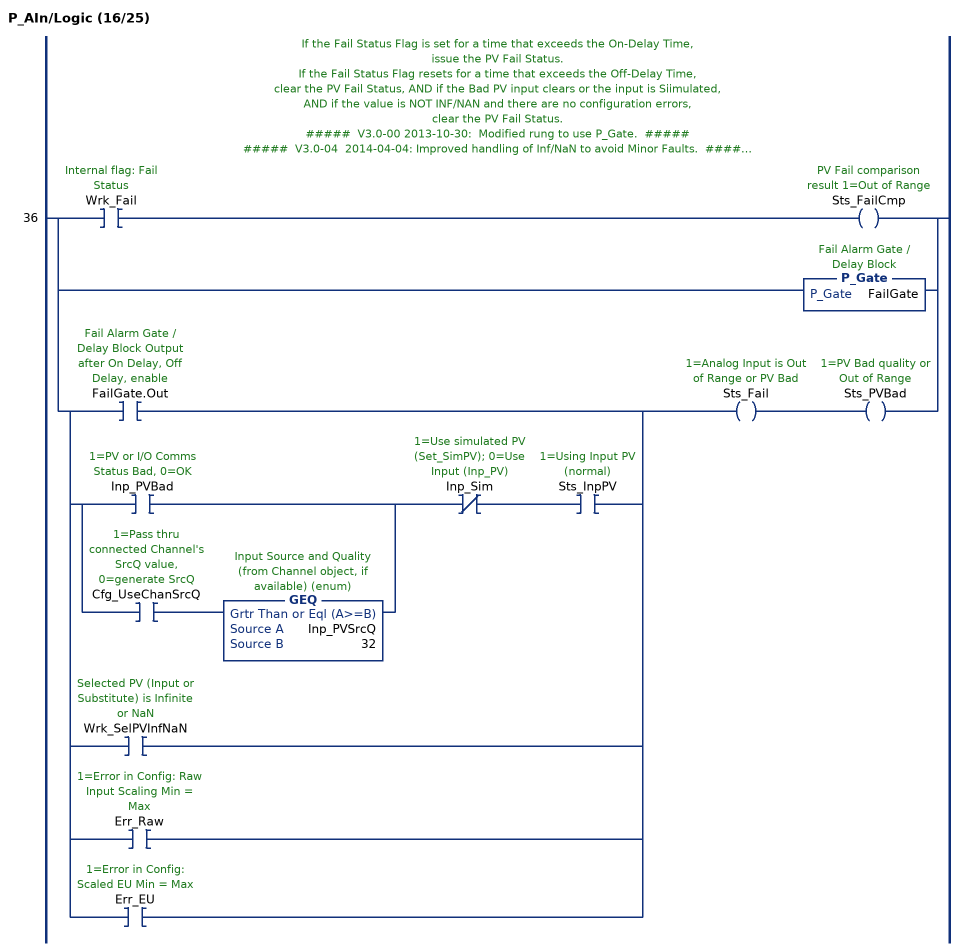
   // If the Fail Status Flag is set for a time that exceeds the On-Delay Time,
   // issue the PV Fail Status.
   // If the Fail Status Flag resets for a time that exceeds the Off-Delay Time,
   // clear the PV Fail Status, AND if the Bad PV input clears or the input is Siimulated,
   // AND if the value is NOT INF/NAN and there are no configuration errors,
   // clear the PV Fail Status.
   // #####  V3.0-00 2013-10-30:  Modified rung to use P_Gate.  #####
   // #####  V3.0-04  2014-04-04: Improved handling of Inf/NaN to avoid Minor Faults.  #####
   // #####  V3.1-00  2014-06-30:  Modified to use input channel Source/Quality enumeration.  #####
   // #####  V3.5-02  2016-03-28:  Modified to add Cfg_UseChanSrcQ.  #####
   36: [XIC(Wrk_Fail) OTE(Sts_FailCmp) ,P_Gate(FailGate) ,[XIC(FailGate.Out) ,[XIC(Inp_PVBad) ,XIC(Cfg_UseChanSrcQ) GEQ(Inp_PVSrcQ,32) ] XIO(Inp_Sim) XIC(Sts_InpPV) ,XIC(Wrk_SelPVInfNaN) ,XIC(Err_Raw) ,XIC(Err_EU) ] OTE(Sts_Fail) OTE(Sts_PVBad) ];
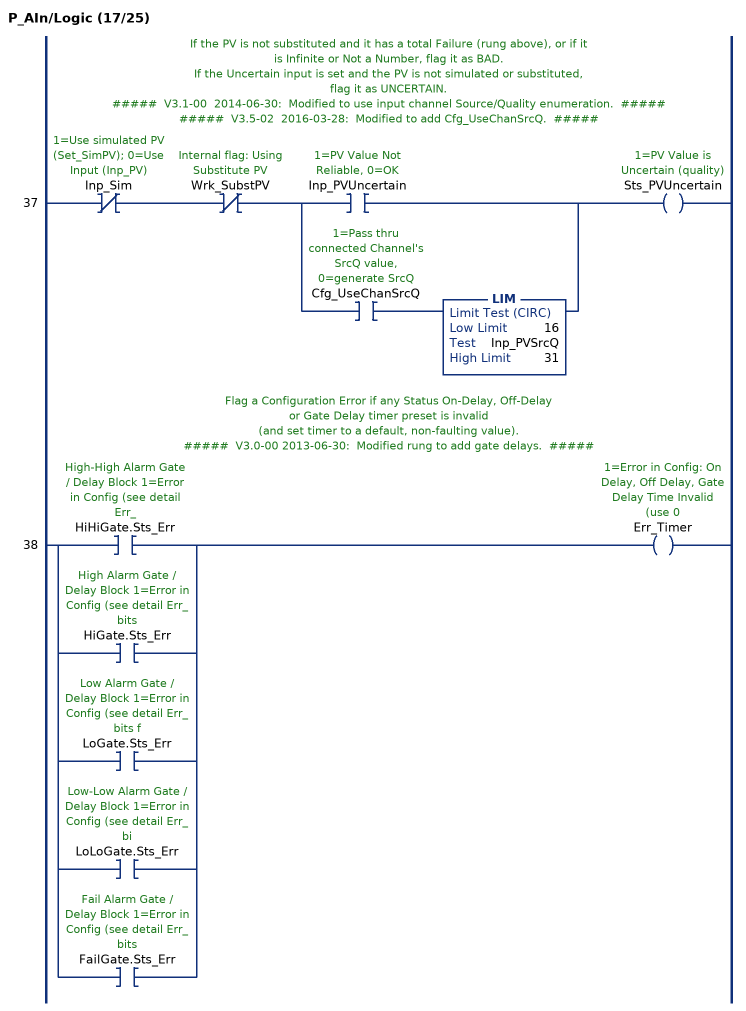
   // If the PV is not substituted and it has a total Failure (rung above), or if it
   // is Infinite or Not a Number, flag it as BAD.
   // If the Uncertain input is set and the PV is not simulated or substituted,
   // flag it as UNCERTAIN.
   // #####  V3.1-00  2014-06-30:  Modified to use input channel Source/Quality enumeration.  #####
   // #####  V3.5-02  2016-03-28:  Modified to add Cfg_UseChanSrcQ.  #####
   37: XIO(Inp_Sim)XIO(Wrk_SubstPV)[XIC(Inp_PVUncertain) ,XIC(Cfg_UseChanSrcQ) LIM(16,Inp_PVSrcQ,31) ]OTE(Sts_PVUncertain);
   // Flag a Configuration Error if any Status On-Delay, Off-Delay
   // or Gate Delay timer preset is invalid
   // (and set timer to a default, non-faulting value).
   // #####  V3.0-00 2013-06-30:  Modified rung to add gate delays.  #####
   38: [XIC(HiHiGate.Sts_Err) ,XIC(HiGate.Sts_Err) ,XIC(LoGate.Sts_Err) ,XIC(LoLoGate.Sts_Err) ,XIC(FailGate.Sts_Err) ]OTE(Err_Timer);
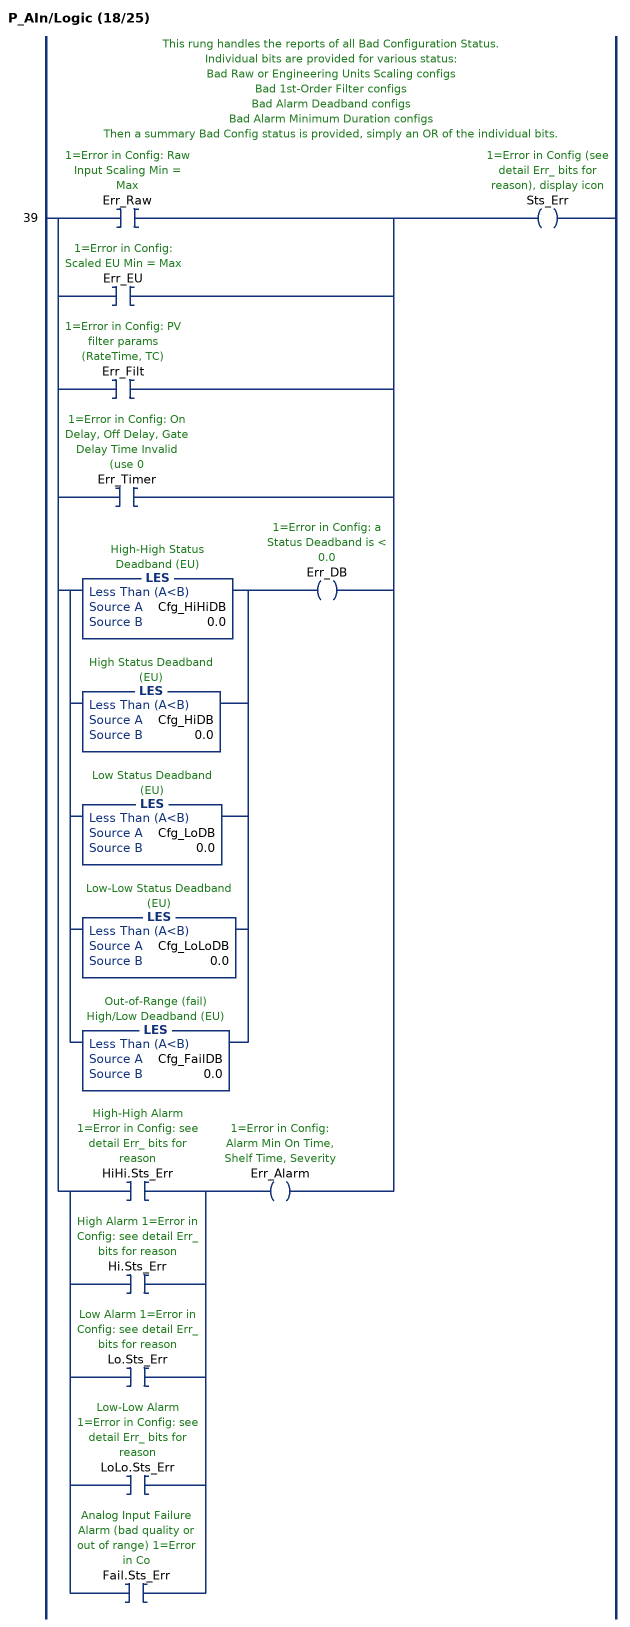
   // This rung handles the reports of all Bad Configuration Status.
   // Individual bits are provided for various status:
   // Bad Raw or Engineering Units Scaling configs
   // Bad 1st-Order Filter configs
   // Bad Alarm Deadband configs
   // Bad Alarm Minimum Duration configs
   // Then a summary Bad Config status is provided, simply an OR of the individual bits.
   39: [XIC(Err_Raw) ,XIC(Err_EU) ,XIC(Err_Filt) ,XIC(Err_Timer) ,[LES(Cfg_HiHiDB,0.0) ,LES(Cfg_HiDB,0.0) ,LES(Cfg_LoDB,0.0) ,LES(Cfg_LoLoDB,0.0) ,LES(Cfg_FailDB,0.0) ] OTE(Err_DB) ,[XIC(HiHi.Sts_Err) ,XIC(Hi.Sts_Err) ,XIC(Lo.Sts_Err) ,XIC(LoLo.Sts_Err) ,XIC(Fail.Sts_Err) ] OTE(Err_Alarm) ]OTE(Sts_Err);
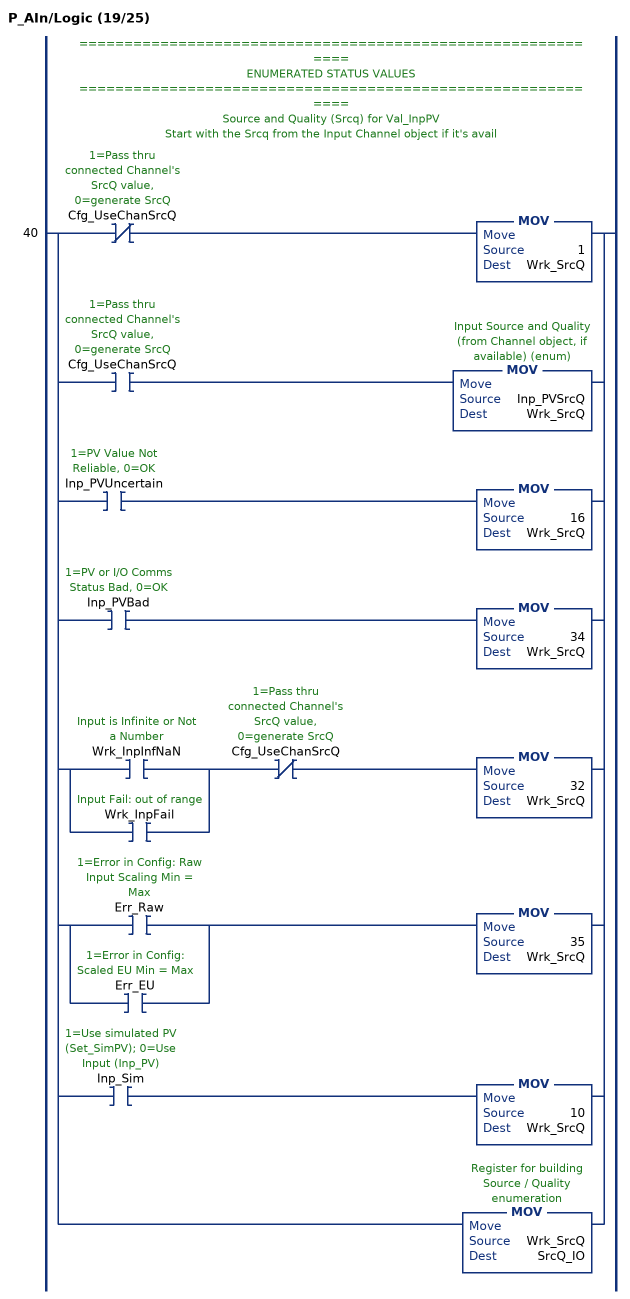
   // ============================================================
   // ENUMERATED STATUS VALUES
   // ============================================================
   // Source and Quality (Srcq) for Val_InpPV
   // Start with the Srcq from the Input Channel object if it's avail
   40: [XIO(Cfg_UseChanSrcQ) MOV(1,Wrk_SrcQ) ,XIC(Cfg_UseChanSrcQ) MOV(Inp_PVSrcQ,Wrk_SrcQ) ,XIC(Inp_PVUncertain) MOV(16,Wrk_SrcQ) ,XIC(Inp_PVBad) MOV(34,Wrk_SrcQ) ,[XIC(Wrk_InpInfNaN) ,XIC(Wrk_InpFail) ] XIO(Cfg_UseChanSrcQ) MOV(32,Wrk_SrcQ) ,[XIC(Err_Raw) ,XIC(Err_EU) ] MOV(35,Wrk_SrcQ) ,XIC(Inp_Sim) MOV(10,Wrk_SrcQ) ,MOV(Wrk_SrcQ,SrcQ_IO) ];
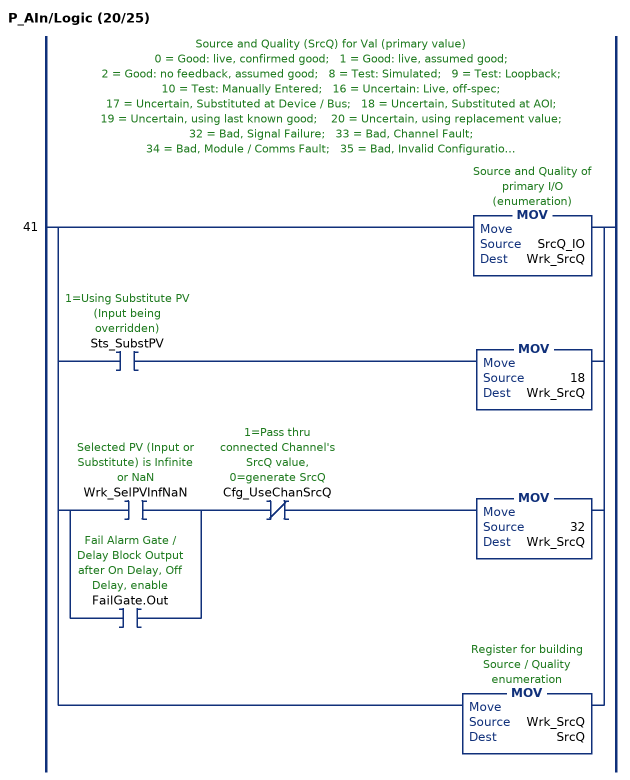
   // Source and Quality (SrcQ) for Val (primary value)
   // 0 = Good: live, confirmed good;   1 = Good: live, assumed good;
   // 2 = Good: no feedback, assumed good;   8 = Test: Simulated;   9 = Test: Loopback;
   // 10 = Test: Manually Entered;   16 = Uncertain: Live, off-spec;
   // 17 = Uncertain, Substituted at Device / Bus;   18 = Uncertain, Substituted at AOI;
   // 19 = Uncertain, using last known good;    20 = Uncertain, using replacement value;
   // 32 = Bad, Signal Failure;   33 = Bad, Channel Fault;
   // 34 = Bad, Module / Comms Fault;   35 = Bad, Invalid Configuration
   // #####  V3.1-00  2014-06-30:  Added rung for Source/Quality enumerations.  #####
   // #####  V3.5-02  2016-03-28:  Modified to add Cfg_UseChanSrcQ.  #####
   41: [MOV(SrcQ_IO,Wrk_SrcQ) ,XIC(Sts_SubstPV) MOV(18,Wrk_SrcQ) ,[XIC(Wrk_SelPVInfNaN) ,XIC(FailGate.Out) ] XIO(Cfg_UseChanSrcQ) MOV(32,Wrk_SrcQ) ,MOV(Wrk_SrcQ,SrcQ) ];
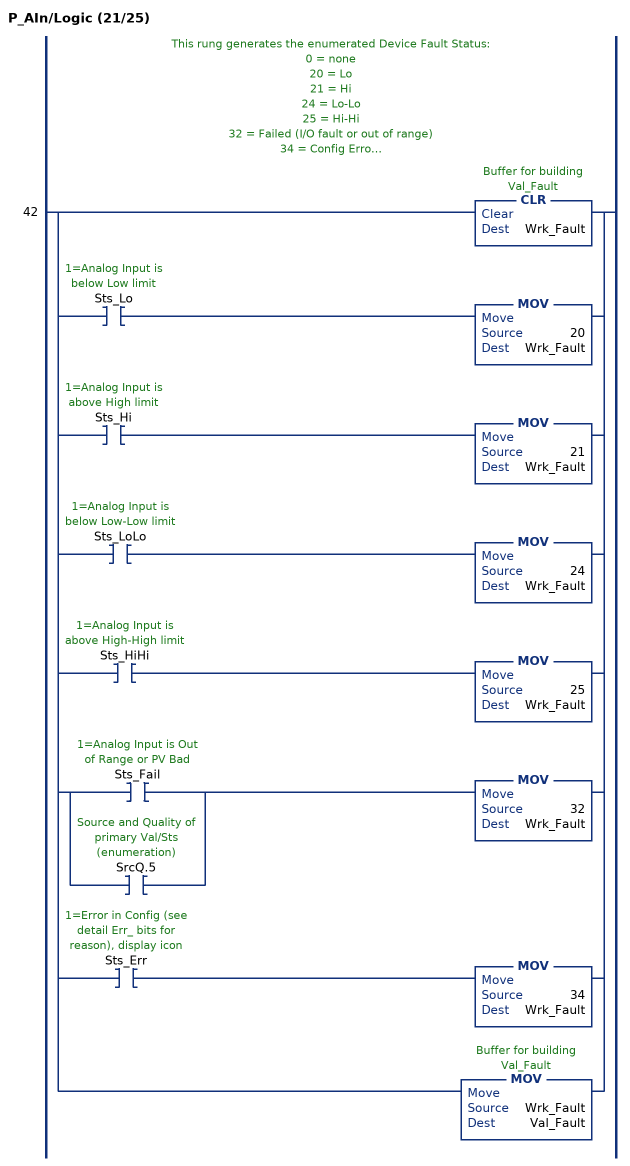
   // This rung generates the enumerated Device Fault Status:
   // 0 = none
   // 20 = Lo
   // 21 = Hi
   // 24 = Lo-Lo
   // 25 = Hi-Hi
   // 32 = Failed (I/O fault or out of range)
   // 34 = Config Error
   // #####  V3.1-05  2016-01-22:  Added check of SrcQ >= 32 for Val_Fault.  #####
   42: [CLR(Wrk_Fault) ,XIC(Sts_Lo) MOV(20,Wrk_Fault) ,XIC(Sts_Hi) MOV(21,Wrk_Fault) ,XIC(Sts_LoLo) MOV(24,Wrk_Fault) ,XIC(Sts_HiHi) MOV(25,Wrk_Fault) ,[XIC(Sts_Fail) ,XIC(SrcQ.5) ] MOV(32,Wrk_Fault) ,XIC(Sts_Err) MOV(34,Wrk_Fault) ,MOV(Wrk_Fault,Val_Fault) ];
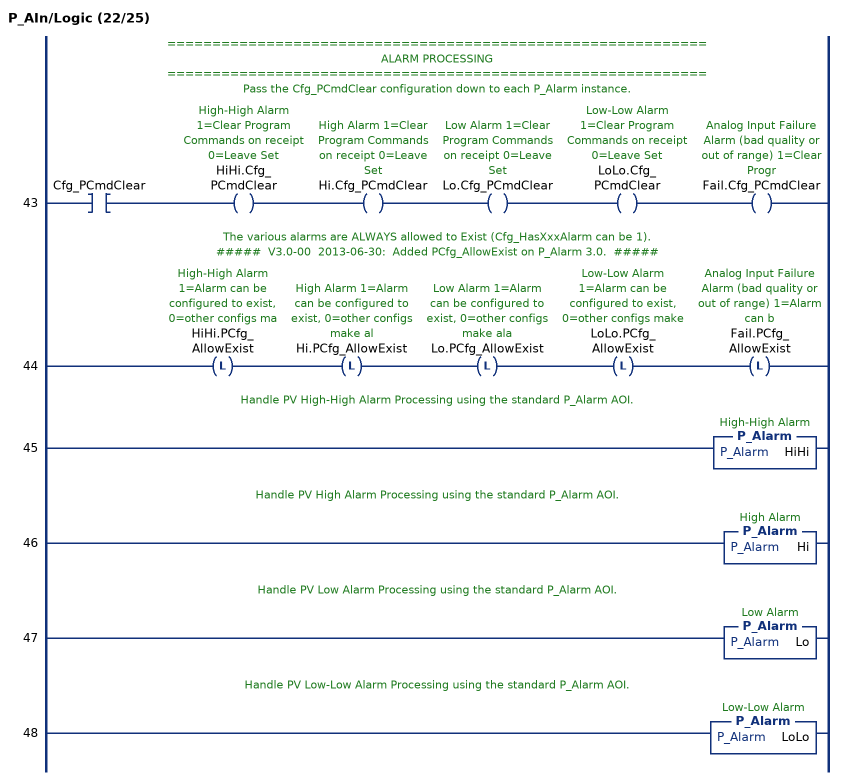
   // ============================================================
   // ALARM PROCESSING
   // ============================================================
   // Pass the Cfg_PCmdClear configuration down to each P_Alarm instance.
   43: XIC(Cfg_PCmdClear)OTE(HiHi.Cfg_PCmdClear)OTE(Hi.Cfg_PCmdClear)OTE(Lo.Cfg_PCmdClear)OTE(LoLo.Cfg_PCmdClear)OTE(Fail.Cfg_PCmdClear);
   // The various alarms are ALWAYS allowed to Exist (Cfg_HasXxxAlarm can be 1).
   // #####  V3.0-00  2013-06-30:  Added PCfg_AllowExist on P_Alarm 3.0.  #####
   44: OTL(HiHi.PCfg_AllowExist)OTL(Hi.PCfg_AllowExist)OTL(Lo.PCfg_AllowExist)OTL(LoLo.PCfg_AllowExist)OTL(Fail.PCfg_AllowExist);
   // Handle PV High-High Alarm Processing using the standard P_Alarm AOI.
   45: P_Alarm(HiHi);
   // Handle PV High Alarm Processing using the standard P_Alarm AOI.
   46: P_Alarm(Hi);
   // Handle PV Low Alarm Processing using the standard P_Alarm AOI.
   47: P_Alarm(Lo);
   // Handle PV Low-Low Alarm Processing using the standard P_Alarm AOI.
   48: P_Alarm(LoLo);
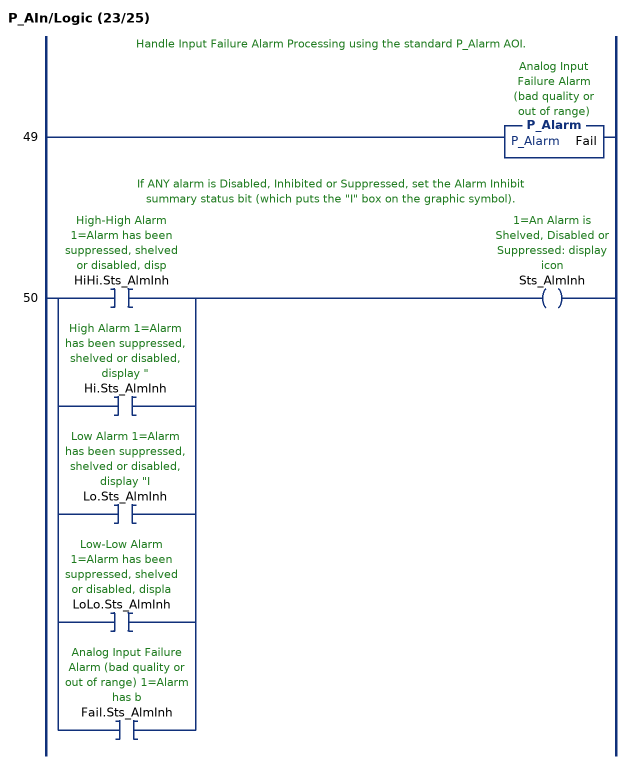
   // Handle Input Failure Alarm Processing using the standard P_Alarm AOI.
   49: P_Alarm(Fail);
   // If ANY alarm is Disabled, Inhibited or Suppressed, set the Alarm Inhibit
   // summary status bit (which puts the "I" box on the graphic symbol).
   50: [XIC(HiHi.Sts_AlmInh) ,XIC(Hi.Sts_AlmInh) ,XIC(Lo.Sts_AlmInh) ,XIC(LoLo.Sts_AlmInh) ,XIC(Fail.Sts_AlmInh) ]OTE(Sts_AlmInh);
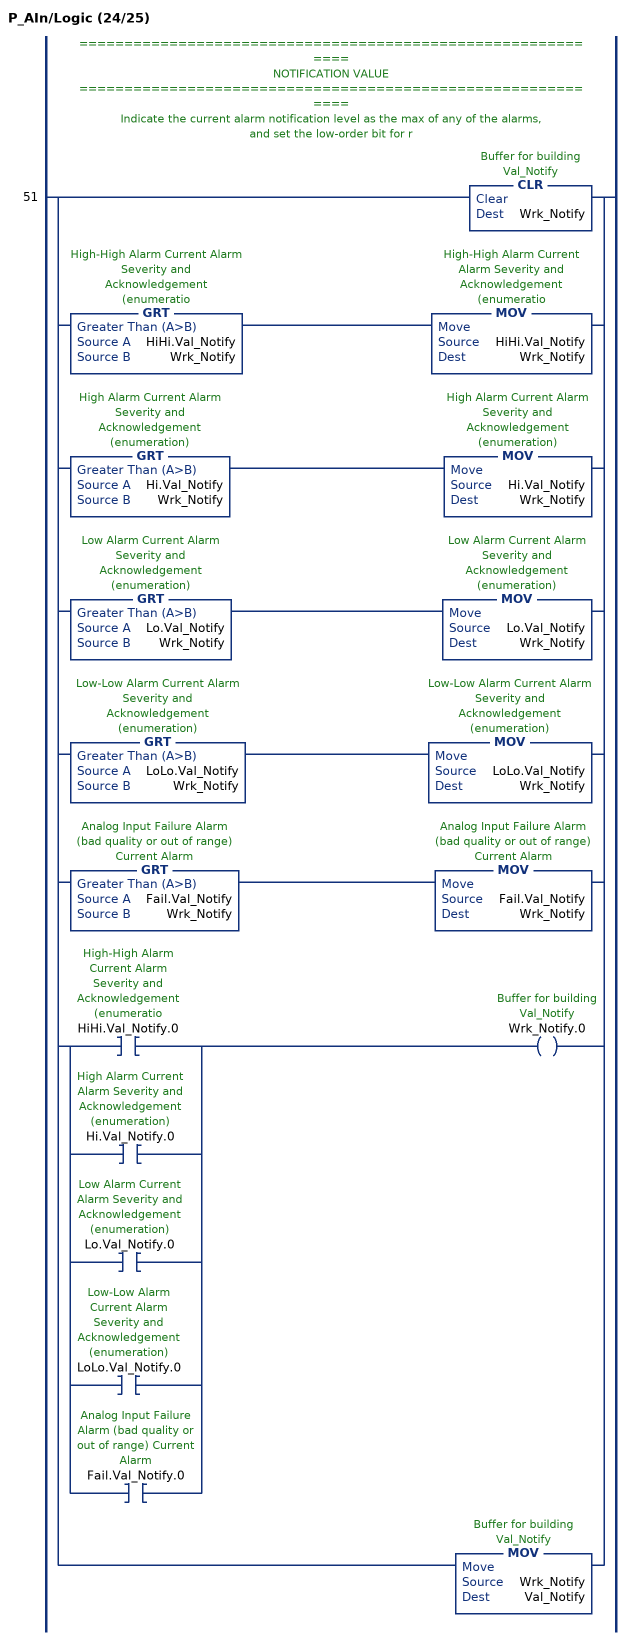
   // ============================================================
   // NOTIFICATION VALUE
   // ============================================================
   // Indicate the current alarm notification level as the max of any of the alarms,
   // and set the low-order bit for r
   51: [CLR(Wrk_Notify) ,GRT(HiHi.Val_Notify,Wrk_Notify) MOV(HiHi.Val_Notify,Wrk_Notify) ,GRT(Hi.Val_Notify,Wrk_Notify) MOV(Hi.Val_Notify,Wrk_Notify) ,GRT(Lo.Val_Notify,Wrk_Notify) MOV(Lo.Val_Notify,Wrk_Notify) ,GRT(LoLo.Val_Notify,Wrk_Notify) MOV(LoLo.Val_Notify,Wrk_Notify) ,GRT(Fail.Val_Notify,Wrk_Notify) MOV(Fail.Val_Notify,Wrk_Notify) ,[XIC(HiHi.Val_Notify.0) ,XIC(Hi.Val_Notify.0) ,XIC(Lo.Val_Notify.0) ,XIC(LoLo.Val_Notify.0) ,XIC(Fail.Val_Notify.0) ] OTE(Wrk_Notify.0) ,MOV(Wrk_Notify,Val_Notify) ];
